KUKA KRL data list: ps_p13060r5_msr_lta_c1.dat

&ACCESS RVO
&REL 5
&COMMENT SOLDA MSR LTA GUN C1
&PARAM DISKPATH = KRC:\R1\Program
DEFDAT  ps_p13060r5_msr_lta_c1
;FOLD EXTERNAL DECLARATIONS;%{PE}%MKUKATPBASIS,%CEXT,%VCOMMON,%P
;FOLD GRIPPERTECH EXT
EXT  H50 (INT  :IN,INT  :IN,INT  :IN,GRP_TYP  :IN )
;ENDFOLD (GRIPPERTECH EXT)
;FOLD SPOTTECH EXT
EXT  USERSPOT (S_COMMAND  :IN,SPOT_TYPE  :IN )
;ENDFOLD (SPOTTECH EXT)
;FOLD BASISTECH EXT;%{PE}%MKUKATPBASIS,%CEXT,%VEXT,%P
EXT  BAS (BAS_COMMAND  :IN,REAL  :IN )
DECL INT SUCCESS
;ENDFOLD (BASISTECH EXT)
;FOLD USER EXT;%{E}%MKUKATPUSER,%CEXT,%VEXT,%P
;Make your modifications here

;ENDFOLD (USER EXT)
;ENDFOLD (EXTERNAL DECLARATIONS)

;# ============ START PATH : swp_p13060r5_msr_lta_c1 =============
DECL FDAT Fp75={TOOL_NO 2,BASE_NO 1,IPO_FRAME #BASE,POINT2[] " "}
DECL PDAT PP_OLP2={VEL 100.0,ACC 100.0,APO_DIST 100.0,APO_MODE #CDIS}
DECL E6POS Xp75={X 1303.604,Y -211.761002,Z 2118.72705,A -126.906303,B 65.6848984,C 49.8302002,S 2,T 10}
DECL FDAT Fp76={TOOL_NO 2,BASE_NO 1,IPO_FRAME #BASE,POINT2[] " "}
DECL PDAT PP_OLP3={VEL 100.0,ACC 100.0,APO_DIST 100.0,APO_MODE #CDIS}
DECL E6POS Xp76={X 1729.96497,Y -537.172974,Z 1590.30103,A -75.8211975,B 62.4005013,C 105.7089,S 2,T 11}
DECL FDAT Fp77={TOOL_NO 2,BASE_NO 1,IPO_FRAME #BASE,POINT2[] " "}
DECL PDAT PP_OLP4={VEL 100.0,ACC 100.0,APO_DIST 100.0,APO_MODE #CDIS}
DECL E6POS Xp77={X 2022.47803,Y -785.769104,Z 542.154907,A -89.9998932,B 70.0002136,C 89.9999771,S 2,T 9,E1 0.0,E2 0.0,E3 0.0,E4 0.0,E5 0.0,E6 0.0}
DECL FDAT Fp78={TOOL_NO 2,BASE_NO 1,IPO_FRAME #BASE,POINT2[] " "}
DECL PDAT PP_OLP5={VEL 100.0,ACC 100.0,APO_DIST 100.0,APO_MODE #CDIS}
DECL E6POS Xp78={X 2134.76611,Y -787.281006,Z 490.900208,A -89.9603119,B 69.9023438,C 90.0867233,S 2,T 9,E1 0.0,E2 0.0,E3 0.0,E4 0.0,E5 0.0,E6 0.0}
DECL FDAT Fswp_60_5471={TOOL_NO 2,BASE_NO 1,IPO_FRAME #BASE,POINT2[] " "}
DECL PDAT PP_OLP6={VEL 100.0,ACC 100.0,APO_DIST 0.0}
DECL SPOT_TYPE SS_OLP1={GUN 2,PAIR #FIRST,RETR #CLO,CLO_TM 0,PGNO1 1,PRESS1 1.0,PGNO2 0,PRESS2 0.0}
DECL E6POS Xswp_60_5471={X 2130.88208,Y -795.672913,Z 457.943512,A -90.164978,B 69.9813766,C 89.8283234,S 2,T 9,E1 0.0,E2 0.0,E3 0.0,E4 0.0,E5 0.0,E6 0.0}
DECL FDAT Fp79={TOOL_NO 2,BASE_NO 1,IPO_FRAME #BASE,POINT2[] " "}
DECL PDAT PP_OLP7={VEL 100.0,ACC 100.0,APO_DIST 100.0,APO_MODE #CDIS}
DECL E6POS Xp79={X 2134.00098,Y -785.97699,Z 492.528015,A -90.0,B 70.0,C 90.0,S 2,T 9,E1 0.0,E2 0.0,E3 0.0,E4 0.0,E5 0.0,E6 0.0}
DECL FDAT Fp80={TOOL_NO 2,BASE_NO 1,IPO_FRAME #BASE,POINT2[] " "}
DECL PDAT PP_OLP8={VEL 100.0,ACC 100.0,APO_DIST 100.0,APO_MODE #CDIS}
DECL E6POS Xp80={X 2023.00098,Y -785.97699,Z 492.527008,A -90.0,B 70.0,C 90.0,S 2,T 9}
DECL FDAT Fp81={TOOL_NO 2,BASE_NO 1,IPO_FRAME #BASE,POINT2[] " "}
DECL PDAT PP_OLP9={VEL 100.0,ACC 100.0,APO_DIST 100.0,APO_MODE #CDIS}
DECL E6POS Xp81={X 1849.08496,Y -251.766006,Z 473.174011,A -153.737396,B 79.8789978,C 25.6958008,S 2,T 9}
DECL FDAT Fp82={TOOL_NO 2,BASE_NO 1,IPO_FRAME #BASE,POINT2[] " "}
DECL PDAT PP_OLP10={VEL 100.0,ACC 100.0,APO_DIST 100.0,APO_MODE #CDIS}
DECL E6POS Xp82={X 2015.50195,Y 281.194,Z 494.32901,A 90.0,B 65.0,C -90.0,S 2,T 33}
DECL FDAT Fp83={TOOL_NO 2,BASE_NO 1,IPO_FRAME #BASE,POINT2[] " "}
DECL PDAT PP_OLP11={VEL 100.0,ACC 100.0,APO_DIST 100.0,APO_MODE #CDIS}
DECL E6POS Xp83={X 2125.00098,Y 281.194,Z 494.32901,A 90.0,B 65.0,C -90.0,S 2,T 33}
DECL FDAT Fswp_60_5452={TOOL_NO 2,BASE_NO 1,IPO_FRAME #BASE,POINT2[] " "}
DECL PDAT PP_OLP12={VEL 100.0,ACC 100.0,APO_DIST 0.0}
DECL SPOT_TYPE SS_OLP2={GUN 1,PAIR #FIRST,RETR #CLO,CLO_TM 0,PGNO1 1,PRESS1 1.0,PGNO2 0,PRESS2 0.0}
DECL E6POS Xswp_60_5452={X 2116.53296,Y 312.069702,Z 459.115387,A 89.9984131,B 64.9997482,C -90.001503,S 2,T 33,E1 0.0,E2 0.0,E3 0.0,E4 0.0,E5 0.0,E6 0.0}
DECL FDAT Fp84={TOOL_NO 2,BASE_NO 1,IPO_FRAME #BASE,POINT2[] " "}
DECL PDAT PP_OLP13={VEL 100.0,ACC 100.0,APO_DIST 100.0,APO_MODE #CDIS}
DECL E6POS Xp84={X 2125.00098,Y 281.194,Z 494.32901,A 90.0,B 65.0,C -90.0,S 2,T 33}
DECL FDAT Fp85={TOOL_NO 2,BASE_NO 1,IPO_FRAME #BASE,POINT2[] " "}
DECL PDAT PP_OLP14={VEL 100.0,ACC 100.0,APO_DIST 100.0,APO_MODE #CDIS}
DECL E6POS Xp85={X 2015.50195,Y 281.194,Z 494.32901,A 90.0,B 65.0,C -90.0,S 2,T 33}
DECL FDAT Fp86={TOOL_NO 2,BASE_NO 1,IPO_FRAME #BASE,POINT2[] " "}
DECL PDAT PP_OLP15={VEL 100.0,ACC 100.0,APO_DIST 100.0,APO_MODE #CDIS}
DECL E6POS Xp86={X 1729.96497,Y 537.172974,Z 1590.30103,A 75.8211975,B 62.4005013,C -105.7089,S 2,T 34}
DECL FDAT Fp87={TOOL_NO 2,BASE_NO 1,IPO_FRAME #BASE,POINT2[] " "}
DECL PDAT PP_OLP16={VEL 100.0,ACC 100.0,APO_DIST 100.0,APO_MODE #CDIS}
DECL E6POS Xp87={X 1303.604,Y 211.761002,Z 2118.72705,A 126.906303,B 65.6848984,C -49.8302002,S 2,T 35}
DECL PDAT PPDAT2={VEL 100.0,ACC 100.0,APO_DIST 100.0,APO_MODE #CDIS}
DECL E6POS XP2={X 814.124023,Y 41.7988205,Z 3106.80688,A -178.988297,B 40.6093292,C 0.315527499,S 2,T 2,E1 0.0,E2 0.0,E3 0.0,E4 0.0,E5 0.0,E6 0.0}
DECL FDAT FP2={TOOL_NO 2,BASE_NO 1,IPO_FRAME #BASE,POINT2[] " "}
DECL PDAT PPDAT3={VEL 100.0,ACC 100.0,APO_DIST 100.0,APO_MODE #CDIS}
DECL E6POS XP3={X 2614.91089,Y 2529.12793,Z 4644.24902,A 61.9992714,B -36.66222,C 37.742569,S 2,T 42,E1 0.0,E2 0.0,E3 0.0,E4 0.0,E5 0.0,E6 0.0}
DECL FDAT FP3={TOOL_NO 2,BASE_NO 1,IPO_FRAME #BASE,POINT2[] " ",TQ_STATE FALSE}
DECL SPOT_SUGG_T LAST_SPOT={GUN[] "1                       ",RETR_CMD[] "#OPN                    ",CHOISE[] "#FIRST                  ",CLO_TM[] "0                       ",PGNO1[] "1                       ",PRESS1[] "0                       ",PGNO2[] "1                       ",PRESS2[] "0                       ",SPOT_PARAMS[] "NORMAL                  "}
DECL FDAT FHOME2={TOOL_NO 0,BASE_NO 0,IPO_FRAME #BASE,POINT2[] " ",TQ_STATE FALSE}
DECL PDAT PPDAT4={VEL 100.0,ACC 100.0,APO_DIST 100.0,APO_MODE #CDIS}
DECL E6POS XpFresa_05={X 1838.66003,Y 2546.56006,Z 4367.69092,A 105.045502,B -33.6448593,C -0.634051323,S 2,T 2,E1 0.0,E2 0.0,E3 0.0,E4 0.0,E5 0.0,E6 0.0}
DECL FDAT FpFresa_05={TOOL_NO 2,BASE_NO 1,IPO_FRAME #BASE,POINT2[] " ",TQ_STATE FALSE}
DECL PDAT PPDAT5={VEL 100.0,ACC 100.0,APO_DIST 100.0,APO_MODE #CDIS}
DECL E6POS XpFresa_06={X 4058.65503,Y 2091.6001,Z 4393.26904,A 52.5592613,B -34.2167282,C -0.74924773,S 2,T 2,E1 0.0,E2 0.0,E3 0.0,E4 0.0,E5 0.0,E6 0.0}
DECL FDAT FpFresa_06={TOOL_NO 2,BASE_NO 1,IPO_FRAME #BASE,POINT2[] " ",TQ_STATE FALSE}
DECL PDAT PPDAT6={VEL 100.0,ACC 100.0,APO_DIST 100.0,APO_MODE #CDIS}
DECL E6POS XpFresa_07={X 4058.65503,Y 2091.6001,Z 4393.26904,A 52.5592613,B -34.2167282,C -0.74924773,S 2,T 2,E1 0.0,E2 0.0,E3 0.0,E4 0.0,E5 0.0,E6 0.0}
DECL FDAT FpFresa_07={TOOL_NO 2,BASE_NO 1,IPO_FRAME #BASE,POINT2[] " ",TQ_STATE FALSE}
DECL PDAT PPDAT7={VEL 100.0,ACC 100.0,APO_DIST 100.0,APO_MODE #CDIS}
DECL E6POS XpFresa_08={X 1838.66003,Y 2546.56006,Z 4367.69092,A 105.045502,B -33.6448593,C -0.634051323,S 2,T 2,E1 0.0,E2 0.0,E3 0.0,E4 0.0,E5 0.0,E6 0.0}
DECL FDAT FpFresa_08={TOOL_NO 2,BASE_NO 1,IPO_FRAME #BASE,POINT2[] " ",TQ_STATE FALSE}
DECL E6POS XP4={X 3802.31104,Y 2105.88989,Z 4640.2832,A 19.5630798,B -23.7333107,C 61.6030312,S 2,T 42,E1 0.0,E2 0.0,E3 0.0,E4 0.0,E5 0.0,E6 0.0}
DECL FDAT FP4={TOOL_NO 2,BASE_NO 1,IPO_FRAME #BASE,POINT2[] " ",TQ_STATE FALSE}
DECL PDAT PPDAT8={VEL 100.0,ACC 100.0,APO_DIST 5.0,APO_MODE #CDIS}
ENDDAT
